// TIA Portal V16 export
// export: Created 2023-01-04T15:44:10.152329Z, ExportSetting WithDefaults, DisplayName Totally Integrated Automation Portal, DisplayVersion V16, DisplayName TIA Portal Version Control Interface, DisplayVersion V16, DisplayName TIA Portal Openness, DisplayVersion V16, DisplayName STEP 7 Professional, DisplayVersion V16, DisplayName STEP 7 Safety, DisplayVersion V16, DisplayName WinCC Advanced, DisplayVersion V16
VAR_GLOBAL   // PLC tag table "P_N_TRIG"
   PTRIG1 AT %M0.0 : Bool;
   PTRIG2 AT %M0.1 : Bool;
   PTRIG3 AT %M0.2 : Bool;
   PTRIG4 AT %M0.3 : Bool;
   PTRIG5 AT %M0.4 : Bool;
   PTRIG6 AT %M0.5 : Bool;
   PTRIG7 AT %M0.6 : Bool;
   PTRIG8 AT %M0.7 : Bool;
   PTRIG9 AT %M1.0 : Bool;
   PTRIG10 AT %M1.1 : Bool;
   PTRIG11 AT %M1.2 : Bool;
   PTRIG12 AT %M1.3 : Bool;
   PTRIG13 AT %M1.4 : Bool;
   PTRIG14 AT %M1.5 : Bool;
   PTRIG15 AT %M1.6 : Bool;
   PTRIG16 AT %M1.7 : Bool;
   PTRIG17 AT %M2.0 : Bool;
   PTRIG18 AT %M2.1 : Bool;
   PTRIG19 AT %M2.2 : Bool;
   PTRIG20 AT %M2.3 : Bool;
   PTRIG21 AT %M2.4 : Bool;
   PTRIG22 AT %M2.5 : Bool;
   PTRIG23 AT %M2.6 : Bool;
   NTRIG1 AT %M2.7 : Bool;
   NTRIG2 AT %M3.0 : Bool;
   NTRIG3 AT %M3.1 : Bool;
   NTRIG4 AT %M3.2 : Bool;
   NTRIG5 AT %M3.3 : Bool;
   NTRIG6 AT %M3.4 : Bool;
   NTRIG7 AT %M3.5 : Bool;
   NTRIG8 AT %M3.6 : Bool;
   NTRIG9 AT %M3.7 : Bool;
   NTRIG10 AT %M4.0 : Bool;
   NTRIG11 AT %M4.1 : Bool;
   NTRIG12 AT %M4.2 : Bool;
   NTRIG13 AT %M4.3 : Bool;
   NTRIG14 AT %M4.4 : Bool;
   NTRIG15 AT %M4.5 : Bool;
   NTRIG16 AT %M4.6 : Bool;
   NTRIG17 AT %M4.7 : Bool;
   NTRIG18 AT %M5.0 : Bool;
   NTRIG19 AT %M5.1 : Bool;
   NTRIG20 AT %M5.2 : Bool;
   PTRIG24 AT %M5.3 : Bool;
   PTRIG25 AT %M5.4 : Bool;
END_VAR
